TYPE ST_OpcuaStatus :
STRUCT
	input	: ST_OpcuaStatus_in;
	
	{attribute 'OPC.UA.DA.Access' := '1'}
	output	: ST_OpcuaStatus_out;
END_STRUCT
END_TYPE

(* stored: Version 1.1.0.1, ProductVersion 3.1.4024.9
   DUT ST_OpcuaStatus: Id {2310f7d7-56b1-4596-bf08-7e840046af3f} *)
